FUNCTION_BLOCK AI1 (* Composite Function Block Type *)
  (* Standard: 61499-2 *)
  (* Version 0.0, 2018-12-26, 4DIAC-IDE, 4DIAC-Consortium *)
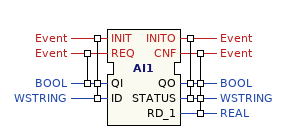
  EVENT_INPUT
    INIT WITH QI, ID; (* Initialization Request *)
    REQ WITH QI; (* Normal Execution Request *)
  END_EVENT
  EVENT_OUTPUT
    INITO WITH QO, STATUS; (* Initialization Confirm *)
    CNF WITH QO, STATUS, RD_1; (* Execution Confirmation *)
  END_EVENT
  VAR_INPUT
    QI : BOOL; (* Input event qualifier *)
    ID : WSTRING;
  END_VAR
  VAR_OUTPUT
    QO : BOOL; (* Output event qualifier *)
    STATUS : WSTRING;
    RD_1 : REAL;
  END_VAR
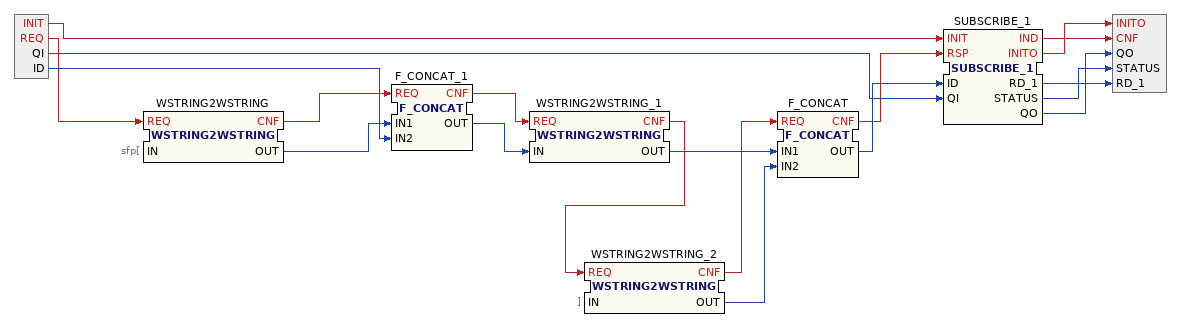
  FBS
    SUBSCRIBE_1 : SUBSCRIBE_1;
    F_CONCAT : F_CONCAT;
    F_CONCAT_1 : F_CONCAT;
    WSTRING2WSTRING : WSTRING2WSTRING(IN := sfp[);
    WSTRING2WSTRING_1 : WSTRING2WSTRING;
    WSTRING2WSTRING_2 : WSTRING2WSTRING(IN := ]);
  END_FBS
  EVENT_CONNECTIONS
    INIT TO SUBSCRIBE_1.INIT;
    F_CONCAT.CNF TO SUBSCRIBE_1.RSP;
    REQ TO WSTRING2WSTRING.REQ;
    WSTRING2WSTRING.CNF TO F_CONCAT_1.REQ;
    F_CONCAT_1.CNF TO WSTRING2WSTRING_1.REQ;
    WSTRING2WSTRING_2.CNF TO F_CONCAT.REQ;
    WSTRING2WSTRING_1.CNF TO WSTRING2WSTRING_2.REQ;
    SUBSCRIBE_1.IND TO CNF;
    SUBSCRIBE_1.INITO TO INITO;
  END_CONNECTIONS
  DATA_CONNECTIONS
    F_CONCAT.OUT TO SUBSCRIBE_1.ID;
    WSTRING2WSTRING.OUT TO F_CONCAT_1.IN1;
    ID TO F_CONCAT_1.IN2;
    QI TO SUBSCRIBE_1.QI;
    F_CONCAT_1.OUT TO WSTRING2WSTRING_1.IN;
    WSTRING2WSTRING_1.OUT TO F_CONCAT.IN1;
    WSTRING2WSTRING_2.OUT TO F_CONCAT.IN2;
    SUBSCRIBE_1.RD_1 TO RD_1;
    SUBSCRIBE_1.STATUS TO STATUS;
    SUBSCRIBE_1.QO TO QO;
  END_CONNECTIONS
END_FUNCTION_BLOCK
